(* PLC project Unnamed, Unknown Unnamed 1 *)
(* stored: creationDateTime 2025-10-27T08:05:43, modificationDateTime 2025-10-27T08:06:42 *)

PROGRAM main

            IF NOT Sensor_Level THEN

    Pump := TRUE;   

    Pump := FALSE; 

END_IF;
          
END_PROGRAM

CONFIGURATION Config0
  RESOURCE Res0 ON PLC
    TASK task0(INTERVAL := T#20ms, PRIORITY := 0);
    PROGRAM instance0 WITH task0 : main;
  END_RESOURCE
END_CONFIGURATION
